// TIA Portal V17 export
// export: Created 2023-09-11T20:22:11.5433454Z, ExportSetting WithDefaults, DisplayName Totally Integrated Automation Portal, DisplayVersion V17 Update 6, DisplayName TIA Portal Openness, DisplayVersion V17 Update 6, DisplayName TIA Portal Teamcenter Gateway, DisplayVersion V17 Update 6, DisplayName TIA Portal Version Control Interface, DisplayVersion V17, DisplayName Simotion SCOUT TIA, DisplayVersion 5.4.3.0, DisplayName TIA Portal Test Suite Advanced, DisplayVersion V17 Update 1, DisplayName SIMOCODE ES, DisplayVersion V17 Update 5, DisplayName SINAMICS Startdrive Advanced, DisplayVersion V17 SP1, DisplayName SINAMICS Startdrive G130, G150, S120, S150, SINAMICS MV, S210, DisplayVersion V17 SP1, DisplayName SINAMICS Startdrive G110M, G120, G120C, G120D, G120P, G115D, DisplayVersion V17 SP1, DisplayName SIRIUS Safety ES, DisplayVersion V17 Update 5, DisplayName STEP 7 Professional, DisplayVersion V17 Update 6, DisplayName STEP 7 CFC, DisplayVersion V17 Update 1, DisplayName STEP 7 Safety, DisplayVersion V17 Update 6, DisplayName WinCC Advanced, DisplayVersion V17 Update 6, DisplayName SIMATIC Visualization Architect, DisplayVersion V17 Update 5
FUNCTION "07_Speed Control" : Void   // FC8, F_LAD
TITLE = Manage Safety Encoder
{ S7_Optimized_Access := 'TRUE' }
VERSION : 0.1
// stored: AutoNumber true, IsIECCheckEnabled false, UDAEnableTagReadback false
BEGIN

REGION Network 1: S1 | =SC01 Upper Coy Sorter
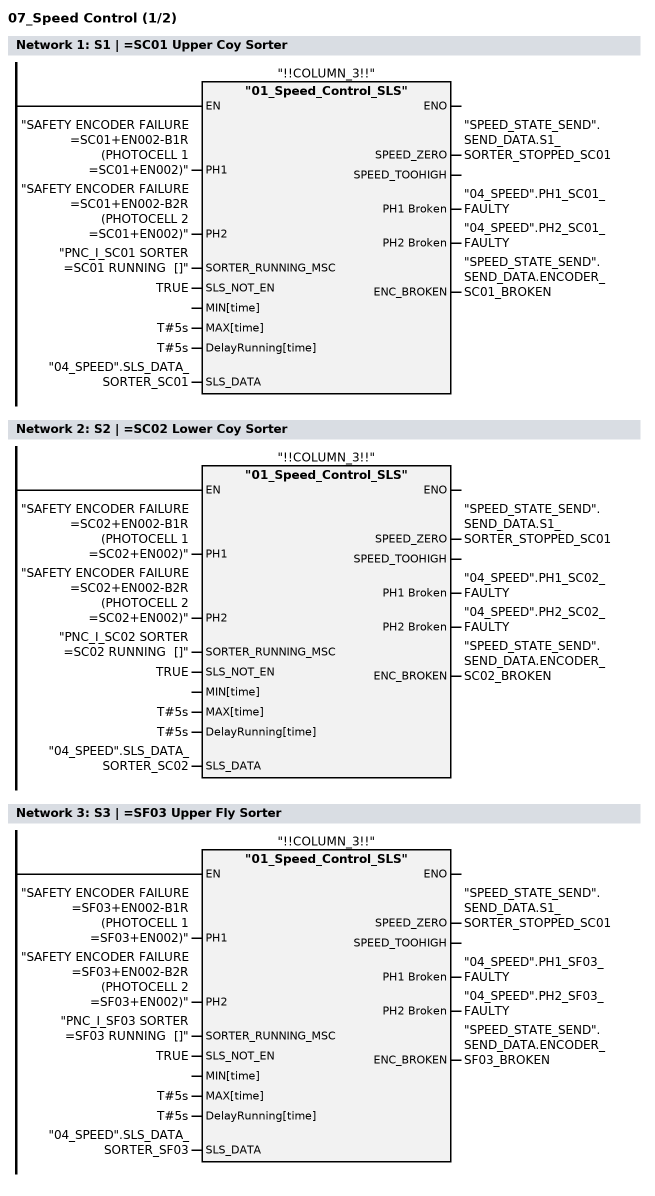
   RUNG wire#powerrail
      "!!COLUMN_3!!"(PH1 := "SAFETY ENCODER FAILURE =SC01+EN002-B1R (PHOTOCELL 1 =SC01+EN002)", PH2 := "SAFETY ENCODER FAILURE =SC01+EN002-B2R (PHOTOCELL 2 =SC01+EN002)", SORTER_RUNNING_MSC := "PNC_I_SC01 SORTER =SC01 RUNNING  []", SLS_NOT_EN := TRUE, "MIN[time]" :=, "MAX[time]" := T#5s, "DelayRunning[time]" := T#5s, SLS_DATA := "04_SPEED".SLS_DATA_SORTER_SC01, SPEED_ZERO => "SPEED_STATE_SEND".SEND_DATA.S1_SORTER_STOPPED_SC01, SPEED_TOOHIGH =>, "PH1 Broken" => "04_SPEED".PH1_SC01_FAULTY, "PH2 Broken" => "04_SPEED".PH2_SC01_FAULTY, ENC_BROKEN => "SPEED_STATE_SEND".SEND_DATA.ENCODER_SC01_BROKEN)
   END_RUNG
   // the same network as SCL:
   "!!COLUMN_3!!"(PH1 := "SAFETY ENCODER FAILURE =SC01+EN002-B1R (PHOTOCELL 1 =SC01+EN002)",   // "01_Speed_Control_SLS"
                  PH2 := "SAFETY ENCODER FAILURE =SC01+EN002-B2R (PHOTOCELL 2 =SC01+EN002)",
                  SORTER_RUNNING_MSC := "PNC_I_SC01 SORTER =SC01 RUNNING  []",
                  SLS_NOT_EN := TRUE,
                  "MAX[time]" := T#5s,
                  "DelayRunning[time]" := T#5s,
                  SLS_DATA := "04_SPEED".SLS_DATA_SORTER_SC01,
                  SPEED_ZERO => "SPEED_STATE_SEND".SEND_DATA.S1_SORTER_STOPPED_SC01,
                  "PH1 Broken" => "04_SPEED".PH1_SC01_FAULTY,
                  "PH2 Broken" => "04_SPEED".PH2_SC01_FAULTY,
                  ENC_BROKEN => "SPEED_STATE_SEND".SEND_DATA.ENCODER_SC01_BROKEN);
END_REGION

REGION Network 2: S2 | =SC02 Lower Coy Sorter
   RUNG wire#powerrail
      "!!COLUMN_3!!"(PH1 := "SAFETY ENCODER FAILURE =SC02+EN002-B1R (PHOTOCELL 1 =SC02+EN002)", PH2 := "SAFETY ENCODER FAILURE =SC02+EN002-B2R (PHOTOCELL 2 =SC02+EN002)", SORTER_RUNNING_MSC := "PNC_I_SC02 SORTER =SC02 RUNNING  []", SLS_NOT_EN := TRUE, "MIN[time]" :=, "MAX[time]" := T#5s, "DelayRunning[time]" := T#5s, SLS_DATA := "04_SPEED".SLS_DATA_SORTER_SC02, SPEED_ZERO => "SPEED_STATE_SEND".SEND_DATA.S1_SORTER_STOPPED_SC01, SPEED_TOOHIGH =>, "PH1 Broken" => "04_SPEED".PH1_SC02_FAULTY, "PH2 Broken" => "04_SPEED".PH2_SC02_FAULTY, ENC_BROKEN => "SPEED_STATE_SEND".SEND_DATA.ENCODER_SC02_BROKEN)
   END_RUNG
   // the same network as SCL:
   "!!COLUMN_3!!"(PH1 := "SAFETY ENCODER FAILURE =SC02+EN002-B1R (PHOTOCELL 1 =SC02+EN002)",   // "01_Speed_Control_SLS"
                  PH2 := "SAFETY ENCODER FAILURE =SC02+EN002-B2R (PHOTOCELL 2 =SC02+EN002)",
                  SORTER_RUNNING_MSC := "PNC_I_SC02 SORTER =SC02 RUNNING  []",
                  SLS_NOT_EN := TRUE,
                  "MAX[time]" := T#5s,
                  "DelayRunning[time]" := T#5s,
                  SLS_DATA := "04_SPEED".SLS_DATA_SORTER_SC02,
                  SPEED_ZERO => "SPEED_STATE_SEND".SEND_DATA.S1_SORTER_STOPPED_SC01,
                  "PH1 Broken" => "04_SPEED".PH1_SC02_FAULTY,
                  "PH2 Broken" => "04_SPEED".PH2_SC02_FAULTY,
                  ENC_BROKEN => "SPEED_STATE_SEND".SEND_DATA.ENCODER_SC02_BROKEN);
END_REGION

REGION Network 3: S3 | =SF03 Upper Fly Sorter
   RUNG wire#powerrail
      "!!COLUMN_3!!"(PH1 := "SAFETY ENCODER FAILURE =SF03+EN002-B1R (PHOTOCELL 1 =SF03+EN002)", PH2 := "SAFETY ENCODER FAILURE =SF03+EN002-B2R (PHOTOCELL 2 =SF03+EN002)", SORTER_RUNNING_MSC := "PNC_I_SF03 SORTER =SF03 RUNNING  []", SLS_NOT_EN := TRUE, "MIN[time]" :=, "MAX[time]" := T#5s, "DelayRunning[time]" := T#5s, SLS_DATA := "04_SPEED".SLS_DATA_SORTER_SF03, SPEED_ZERO => "SPEED_STATE_SEND".SEND_DATA.S1_SORTER_STOPPED_SC01, SPEED_TOOHIGH =>, "PH1 Broken" => "04_SPEED".PH1_SF03_FAULTY, "PH2 Broken" => "04_SPEED".PH2_SF03_FAULTY, ENC_BROKEN => "SPEED_STATE_SEND".SEND_DATA.ENCODER_SF03_BROKEN)
   END_RUNG
   // the same network as SCL:
   "!!COLUMN_3!!"(PH1 := "SAFETY ENCODER FAILURE =SF03+EN002-B1R (PHOTOCELL 1 =SF03+EN002)",   // "01_Speed_Control_SLS"
                  PH2 := "SAFETY ENCODER FAILURE =SF03+EN002-B2R (PHOTOCELL 2 =SF03+EN002)",
                  SORTER_RUNNING_MSC := "PNC_I_SF03 SORTER =SF03 RUNNING  []",
                  SLS_NOT_EN := TRUE,
                  "MAX[time]" := T#5s,
                  "DelayRunning[time]" := T#5s,
                  SLS_DATA := "04_SPEED".SLS_DATA_SORTER_SF03,
                  SPEED_ZERO => "SPEED_STATE_SEND".SEND_DATA.S1_SORTER_STOPPED_SC01,
                  "PH1 Broken" => "04_SPEED".PH1_SF03_FAULTY,
                  "PH2 Broken" => "04_SPEED".PH2_SF03_FAULTY,
                  ENC_BROKEN => "SPEED_STATE_SEND".SEND_DATA.ENCODER_SF03_BROKEN);
END_REGION

REGION Network 4: S4 | =SF04 Lower Fly Sorter
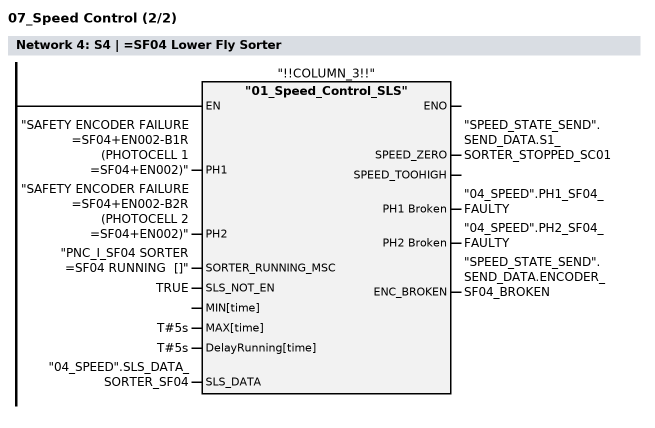
   RUNG wire#powerrail
      "!!COLUMN_3!!"(PH1 := "SAFETY ENCODER FAILURE =SF04+EN002-B1R (PHOTOCELL 1 =SF04+EN002)", PH2 := "SAFETY ENCODER FAILURE =SF04+EN002-B2R (PHOTOCELL 2 =SF04+EN002)", SORTER_RUNNING_MSC := "PNC_I_SF04 SORTER =SF04 RUNNING  []", SLS_NOT_EN := TRUE, "MIN[time]" :=, "MAX[time]" := T#5s, "DelayRunning[time]" := T#5s, SLS_DATA := "04_SPEED".SLS_DATA_SORTER_SF04, SPEED_ZERO => "SPEED_STATE_SEND".SEND_DATA.S1_SORTER_STOPPED_SC01, SPEED_TOOHIGH =>, "PH1 Broken" => "04_SPEED".PH1_SF04_FAULTY, "PH2 Broken" => "04_SPEED".PH2_SF04_FAULTY, ENC_BROKEN => "SPEED_STATE_SEND".SEND_DATA.ENCODER_SF04_BROKEN)
   END_RUNG
   // the same network as SCL:
   "!!COLUMN_3!!"(PH1 := "SAFETY ENCODER FAILURE =SF04+EN002-B1R (PHOTOCELL 1 =SF04+EN002)",   // "01_Speed_Control_SLS"
                  PH2 := "SAFETY ENCODER FAILURE =SF04+EN002-B2R (PHOTOCELL 2 =SF04+EN002)",
                  SORTER_RUNNING_MSC := "PNC_I_SF04 SORTER =SF04 RUNNING  []",
                  SLS_NOT_EN := TRUE,
                  "MAX[time]" := T#5s,
                  "DelayRunning[time]" := T#5s,
                  SLS_DATA := "04_SPEED".SLS_DATA_SORTER_SF04,
                  SPEED_ZERO => "SPEED_STATE_SEND".SEND_DATA.S1_SORTER_STOPPED_SC01,
                  "PH1 Broken" => "04_SPEED".PH1_SF04_FAULTY,
                  "PH2 Broken" => "04_SPEED".PH2_SF04_FAULTY,
                  ENC_BROKEN => "SPEED_STATE_SEND".SEND_DATA.ENCODER_SF04_BROKEN);
END_REGION
END_FUNCTION
